(* Logix 5000 project; controller KTC_lab7 vendor 1 type 14 code 150 rev 30.11; software revision 30.00 *)

TASK MainTask (continuous, watchdog 500 ms) : MainProgram

MODULES
   Local : vendor 1 type 14 code 150 (Compact 0, rev 30.11)
      Analog_IO : Embedded (Compact 2, rev 1.1, Output RPI 80 ms)
      Counters : Embedded (Compact 3, rev 1.1, Output RPI 20 ms)
      Discrete_IO : Embedded (Compact 1, rev 3.1, Output RPI 20 ms)
END_MODULES

PROGRAM MainProgram   (* main routine MainRoutine *)
VAR
   H_1 : ALIAS FOR Local:1:O.Data.7;   // HORN
   M_1 : ALIAS FOR Local:1:O.Data.3;   // MOTOR
   PB_1 : ALIAS FOR Local:1:I.Data.0;   // START UP
   PB_2 : ALIAS FOR Local:1:I.Data.1;   // RESET
   T4_1 : TIMER := (PRE := 10000);
END_VAR

ROUTINE MainRoutine   (* ladder *)
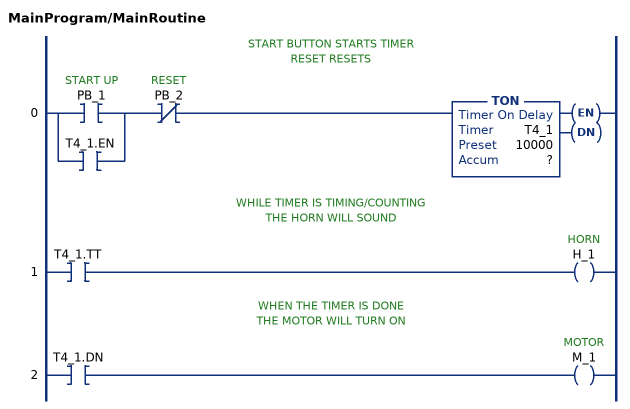
   // START BUTTON STARTS TIMER
   // RESET RESETS
   0: [XIC(PB_1) ,XIC(T4_1.EN) ]XIO(PB_2)TON(T4_1,?,?);
   // WHILE TIMER IS TIMING/COUNTING
   // THE HORN WILL SOUND
   1: XIC(T4_1.TT)OTE(H_1);
   // WHEN THE TIMER IS DONE
   // THE MOTOR WILL TURN ON
   2: XIC(T4_1.DN)OTE(M_1);
END_ROUTINE
END_PROGRAM
